(* PLC project CoDeSys External Library Template, WAGO e!COCKPIT e!COCKPIT, author 3S - Smart Software Solutions GmbH *)
(* stored: creationDateTime 2019-10-29T12:37:19.4786048, version 3.5.5.30, modificationDateTime 2019-10-29T12:36:39.3744516, organization 3S - Smart Software Solutions GmbH *)
(* Library project template with all possible element types, docu and a sample project structure *)

(* values of enumPPPSZadajnikError: BrakKomunikacji: brak komunikacji z zadajnikiem (po EnOcean); AlarmOgolny: alarm ogólny; AlarmCzujnika: alarm braku zmiany wartości czujnika temp. *)

(* Autor: Paweł Kąkol, 2018-08-13-PK Prawa majątkowe: Solwena Sp. z o.o., Aktualizacje: 2019-02-14-AWy - alarm czujnika temperatury Opis: enum służy do obsługi alarmów w fb zadajnika FCP0 na budynkach PPP Sopot *)
{attribute 'qualified_only'}
{attribute 'strict'}
TYPE enumPPPSZadajnikError : (BrakKomunikacji := 1, AlarmOgolny := 2, AlarmCzujnika := 3);
END_TYPE
